// Mitsubishi GX Works2 project: PLC0918_V1   PLC: Q02/Q02H

PROGRAM MAIN
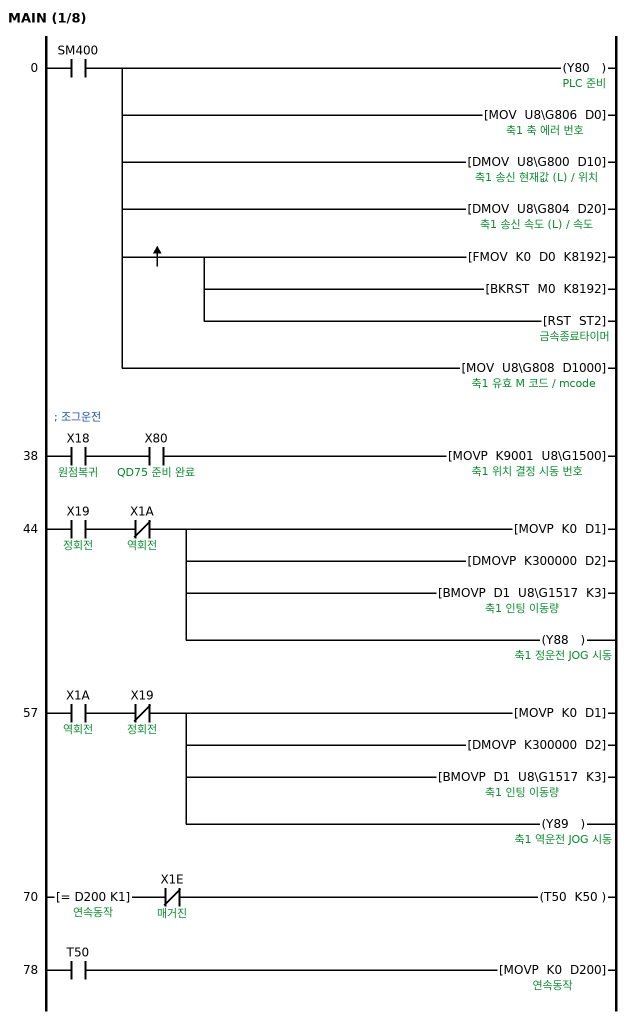
0     LD      SM400
      OUT     Y80  ; PLC 준비
      MOV     U8\G806 D0  ; 축1 축 에러 번호
      DMOV    U8\G800 D10  ; 축1 송신 현재값 (L) / 위치
      DMOV    U8\G804 D20  ; 축1 송신 속도 (L) / 속도
      MPS
      MEP
      FMOV    K0 D0 K8192
      BKRST   M0 K8192
      RST     ST2  ; 금속종료타이머
      MPP
      MOV     U8\G808 D1000  ; 축1 유효 M 코드 / mcode
; 조그운전
38    LD      X18  ; 원점복귀
      AND     X80  ; QD75 준비 완료
      MOVP    K9001 U8\G1500  ; 축1 위치 결정 시동 번호
44    LD      X19  ; 정회전
      ANI     X1A  ; 역회전
      MOVP    K0 D1
      DMOVP   K300000 D2
      BMOVP   D1 U8\G1517 K3  ; 축1 인팅 이동량
      OUT     Y88  ; 축1 정운전 JOG 시동
57    LD      X1A  ; 역회전
      ANI     X19  ; 정회전
      MOVP    K0 D1
      DMOVP   K300000 D2
      BMOVP   D1 U8\G1517 K3
      OUT     Y89  ; 축1 역운전 JOG 시동
70    LD=     D200 K1  ; 연속동작
      ANI     X1E  ; 매거진
      OUT     T50 K50
78    LD      T50
      MOVP    K0 D200
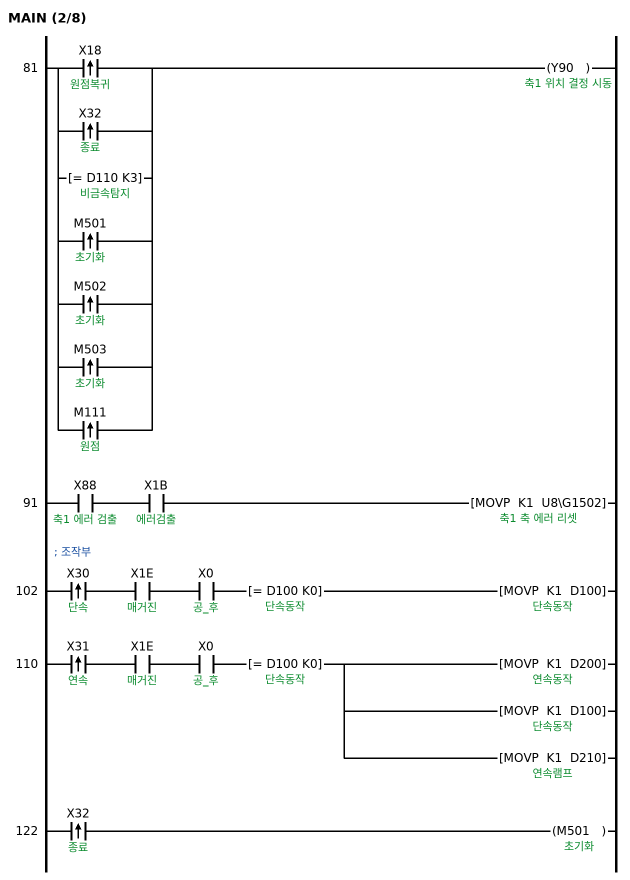
81    LDP     X18  ; 원점복귀
      ORP     X32  ; 종료
      OR=     D110 K3  ; 비금속탐지
      ORP     M501  ; 초기화
      ORP     M502  ; 초기화
      ORP     M503  ; 초기화
      ORP     M111  ; 원점
      OUT     Y90  ; 축1 위치 결정 시동
91    LD      X88  ; 축1 에러 검출
      AND     X1B  ; 에러검출
      MOVP    K1 U8\G1502  ; 축1 축 에러 리셋
; 조작부
102   LDP     X30  ; 단속
      AND     X1E  ; 매거진
      AND     X0  ; 공_후
      AND=    D100 K0  ; 단속동작
      MOVP    K1 D100
110   LDP     X31  ; 연속
      AND     X1E  ; 매거진
      AND     X0  ; 공_후
      AND=    D100 K0  ; 단속동작
      MOVP    K1 D200
      MOVP    K1 D100
      MOVP    K1 D210  ; 연속램프
122   LDP     X32  ; 종료
      OUT     M501  ; 초기화
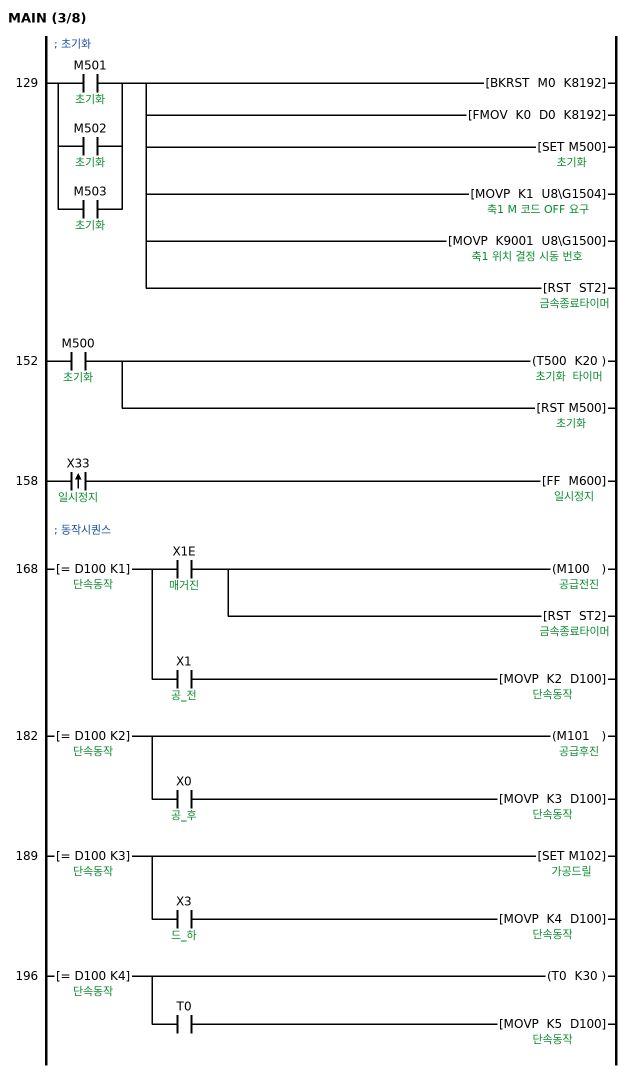
; 초기화
129   LD      M501  ; 초기화
      OR      M502  ; 초기화
      OR      M503  ; 초기화
      BKRST   M0 K8192
      FMOV    K0 D0 K8192
      SET     M500  ; 초기화
      MOVP    K1 U8\G1504  ; 축1 M 코드 OFF 요구
      MOVP    K9001 U8\G1500
      RST     ST2  ; 금속종료타이머
152   LD      M500  ; 초기화
      OUT     T500 K20  ; 초기화  타이머
      RST     M500  ; 초기화
158   LDP     X33  ; 일시정지
      FF      M600  ; 일시정지
; 동작시퀀스
168   LD=     D100 K1  ; 단속동작
      MPS
      AND     X1E  ; 매거진
      OUT     M100  ; 공급전진
      RST     ST2  ; 금속종료타이머
      MPP
      AND     X1  ; 공_전
      MOVP    K2 D100
182   LD=     D100 K2  ; 단속동작
      OUT     M101  ; 공급후진
      AND     X0  ; 공_후
      MOVP    K3 D100
189   LD=     D100 K3  ; 단속동작
      SET     M102  ; 가공드릴
      AND     X3  ; 드_하
      MOVP    K4 D100
196   LD=     D100 K4  ; 단속동작
      OUT     T0 K30
      AND     T0
      MOVP    K5 D100
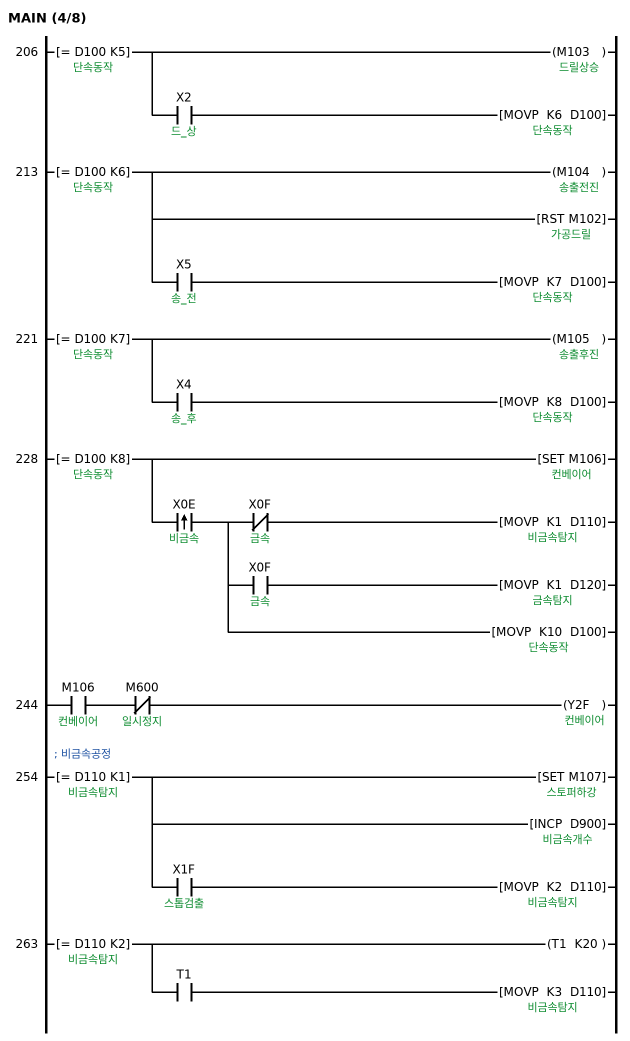
206   LD=     D100 K5  ; 단속동작
      OUT     M103  ; 드릴상승
      AND     X2  ; 드_상
      MOVP    K6 D100
213   LD=     D100 K6  ; 단속동작
      OUT     M104  ; 송출전진
      RST     M102  ; 가공드릴
      AND     X5  ; 송_전
      MOVP    K7 D100
221   LD=     D100 K7  ; 단속동작
      OUT     M105  ; 송출후진
      AND     X4  ; 송_후
      MOVP    K8 D100
228   LD=     D100 K8  ; 단속동작
      SET     M106  ; 컨베이어
      ANDP    X0E  ; 비금속
      MPS
      ANI     X0F  ; 금속
      MOVP    K1 D110
      MRD
      AND     X0F  ; 금속
      MOVP    K1 D120  ; 금속탐지
      MPP
      MOVP    K10 D100
244   LD      M106  ; 컨베이어
      ANI     M600  ; 일시정지
      OUT     Y2F  ; 컨베이어
; 비금속공정
254   LD=     D110 K1  ; 비금속탐지
      SET     M107  ; 스토퍼하강
      INCP    D900  ; 비금속개수
      AND     X1F  ; 스톱검출
      MOVP    K2 D110
263   LD=     D110 K2  ; 비금속탐지
      OUT     T1 K20
      AND     T1
      MOVP    K3 D110
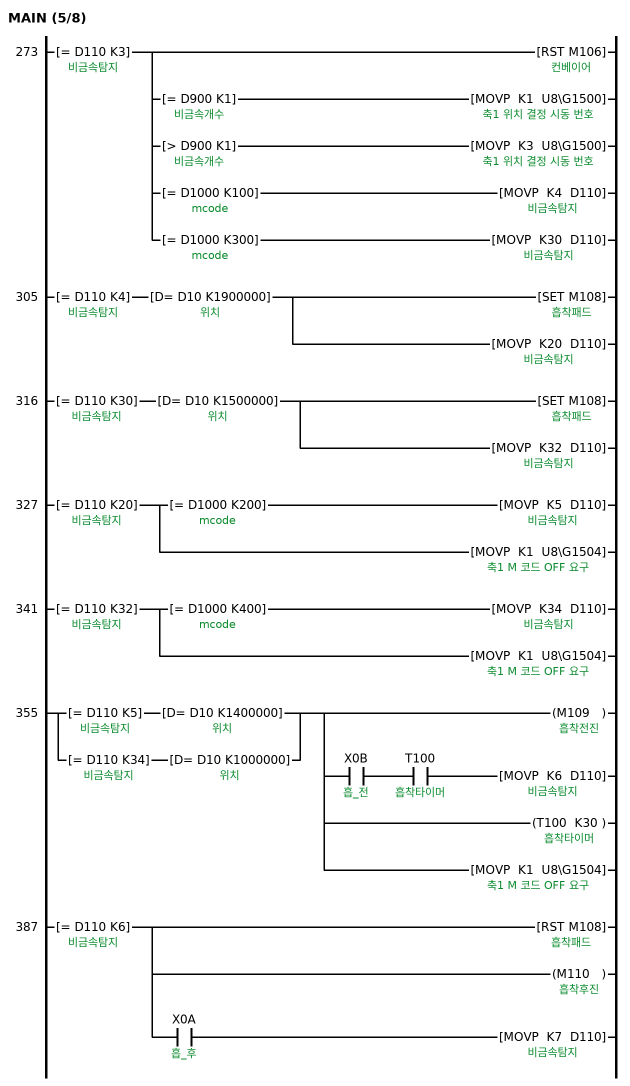
273   LD=     D110 K3  ; 비금속탐지
      RST     M106  ; 컨베이어
      MPS
      AND=    D900 K1  ; 비금속개수
      MOVP    K1 U8\G1500
      MRD
      AND>    D900 K1  ; 비금속개수
      MOVP    K3 U8\G1500
      MRD
      AND=    D1000 K100  ; mcode
      MOVP    K4 D110
      MPP
      AND=    D1000 K300  ; mcode
      MOVP    K30 D110
305   LD=     D110 K4  ; 비금속탐지
      ANDD=   D10 K1900000  ; 위치
      SET     M108  ; 흡착패드
      MOVP    K20 D110
316   LD=     D110 K30  ; 비금속탐지
      ANDD=   D10 K1500000  ; 위치
      SET     M108  ; 흡착패드
      MOVP    K32 D110
327   LD=     D110 K20  ; 비금속탐지
      MPS
      AND=    D1000 K200  ; mcode
      MOVP    K5 D110
      MPP
      MOVP    K1 U8\G1504
341   LD=     D110 K32  ; 비금속탐지
      MPS
      AND=    D1000 K400  ; mcode
      MOVP    K34 D110
      MPP
      MOVP    K1 U8\G1504
355   LD=     D110 K5  ; 비금속탐지
      ANDD=   D10 K1400000  ; 위치
      LD=     D110 K34  ; 비금속탐지
      ANDD=   D10 K1000000  ; 위치
      ORB
      OUT     M109  ; 흡착전진
      MPS
      AND     X0B  ; 흡_전
      AND     T100  ; 흡착타이머
      MOVP    K6 D110
      MPP
      OUT     T100 K30  ; 흡착타이머
      MOVP    K1 U8\G1504
387   LD=     D110 K6  ; 비금속탐지
      RST     M108  ; 흡착패드
      OUT     M110  ; 흡착후진
      AND     X0A  ; 흡_후
      MOVP    K7 D110
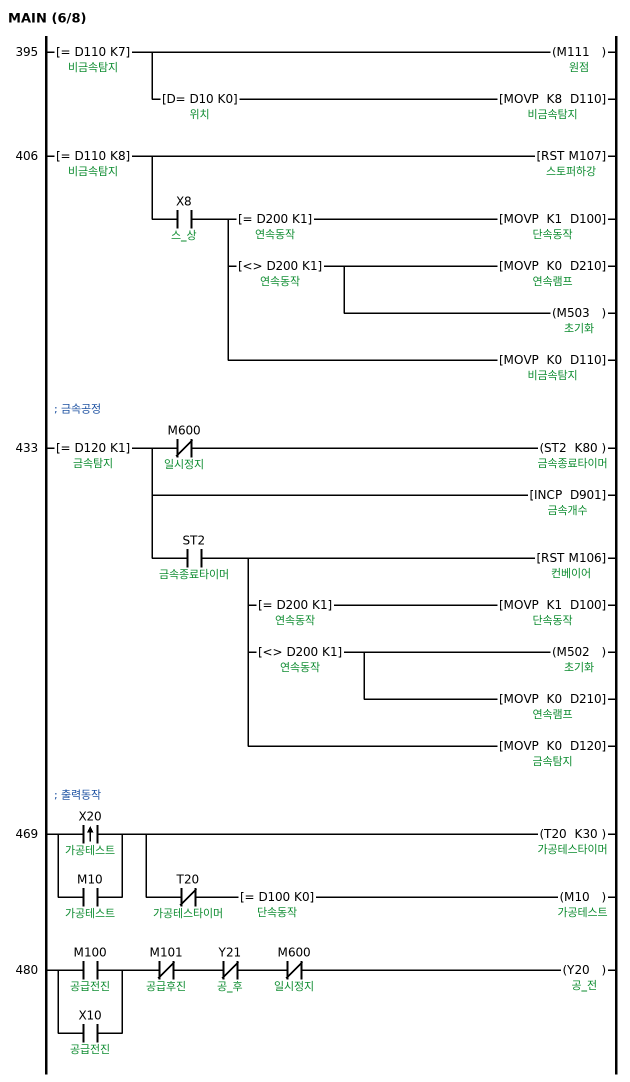
395   LD=     D110 K7  ; 비금속탐지
      OUT     M111  ; 원점
      ANDD=   D10 K0  ; 위치
      MOVP    K8 D110
406   LD=     D110 K8  ; 비금속탐지
      RST     M107  ; 스토퍼하강
      AND     X8  ; 스_상
      MPS
      AND=    D200 K1  ; 연속동작
      MOVP    K1 D100
      MRD
      AND<>   D200 K1  ; 연속동작
      MOVP    K0 D210
      OUT     M503  ; 초기화
      MPP
      MOVP    K0 D110
; 금속공정
433   LD=     D120 K1  ; 금속탐지
      MPS
      ANI     M600  ; 일시정지
      OUT     ST2 K80  ; 금속종료타이머
      MPP
      INCP    D901  ; 금속개수
      AND     ST2  ; 금속종료타이머
      RST     M106  ; 컨베이어
      MPS
      AND=    D200 K1  ; 연속동작
      MOVP    K1 D100
      MRD
      AND<>   D200 K1  ; 연속동작
      OUT     M502  ; 초기화
      MOVP    K0 D210
      MPP
      MOVP    K0 D120
; 출력동작
469   LDP     X20  ; 가공테스트
      OR      M10  ; 가공테스트
      OUT     T20 K30  ; 가공테스타이머
      ANI     T20  ; 가공테스타이머
      AND=    D100 K0  ; 단속동작
      OUT     M10  ; 가공테스트
480   LD      M100  ; 공급전진
      OR      X10  ; 공급전진
      ANI     M101  ; 공급후진
      ANI     Y21  ; 공_후
      ANI     M600  ; 일시정지
      OUT     Y20  ; 공_전
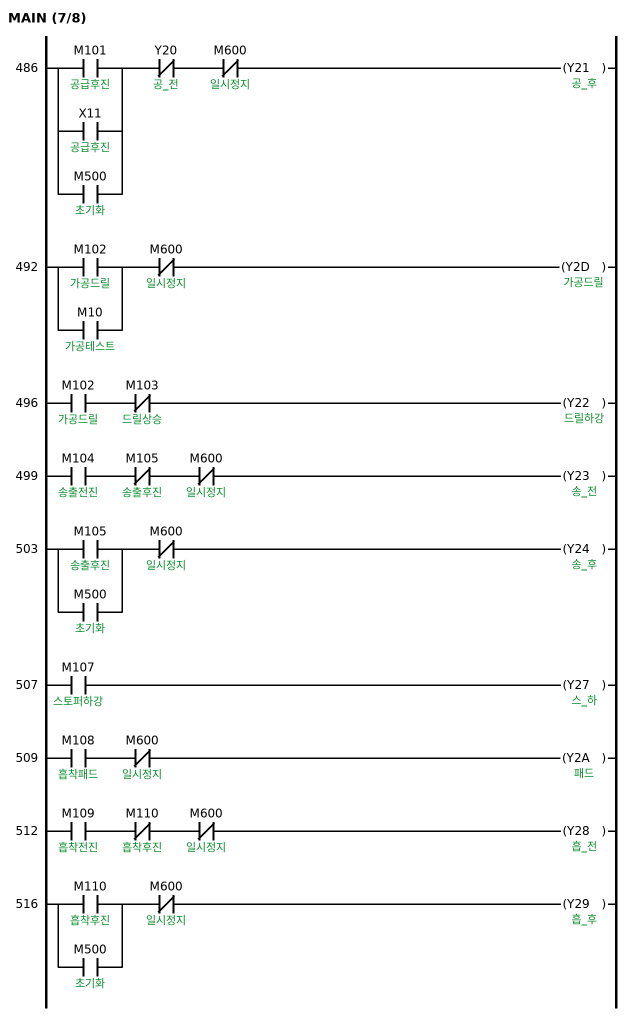
486   LD      M101  ; 공급후진
      OR      X11  ; 공급후진
      OR      M500  ; 초기화
      ANI     Y20  ; 공_전
      ANI     M600  ; 일시정지
      OUT     Y21  ; 공_후
492   LD      M102  ; 가공드릴
      OR      M10  ; 가공테스트
      ANI     M600  ; 일시정지
      OUT     Y2D  ; 가공드릴
496   LD      M102  ; 가공드릴
      ANI     M103  ; 드릴상승
      OUT     Y22  ; 드릴하강
499   LD      M104  ; 송출전진
      ANI     M105  ; 송출후진
      ANI     M600  ; 일시정지
      OUT     Y23  ; 송_전
503   LD      M105  ; 송출후진
      OR      M500  ; 초기화
      ANI     M600  ; 일시정지
      OUT     Y24  ; 송_후
507   LD      M107  ; 스토퍼하강
      OUT     Y27  ; 스_하
509   LD      M108  ; 흡착패드
      ANI     M600  ; 일시정지
      OUT     Y2A  ; 패드
512   LD      M109  ; 흡착전진
      ANI     M110  ; 흡착후진
      ANI     M600  ; 일시정지
      OUT     Y28  ; 흡_전
516   LD      M110  ; 흡착후진
      OR      M500  ; 초기화
      ANI     M600  ; 일시정지
      OUT     Y29  ; 흡_후
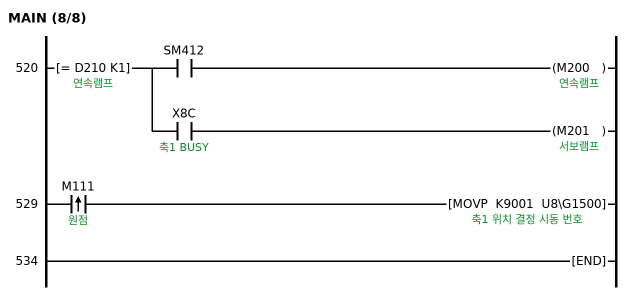
520   LD=     D210 K1  ; 연속램프
      MPS
      AND     SM412
      OUT     M200  ; 연속램프
      MPP
      AND     X8C  ; 축1 BUSY
      OUT     M201  ; 서보램프
529   LDP     M111  ; 원점
      MOVP    K9001 U8\G1500
534   END
END_PROGRAM

PROGRAM test2
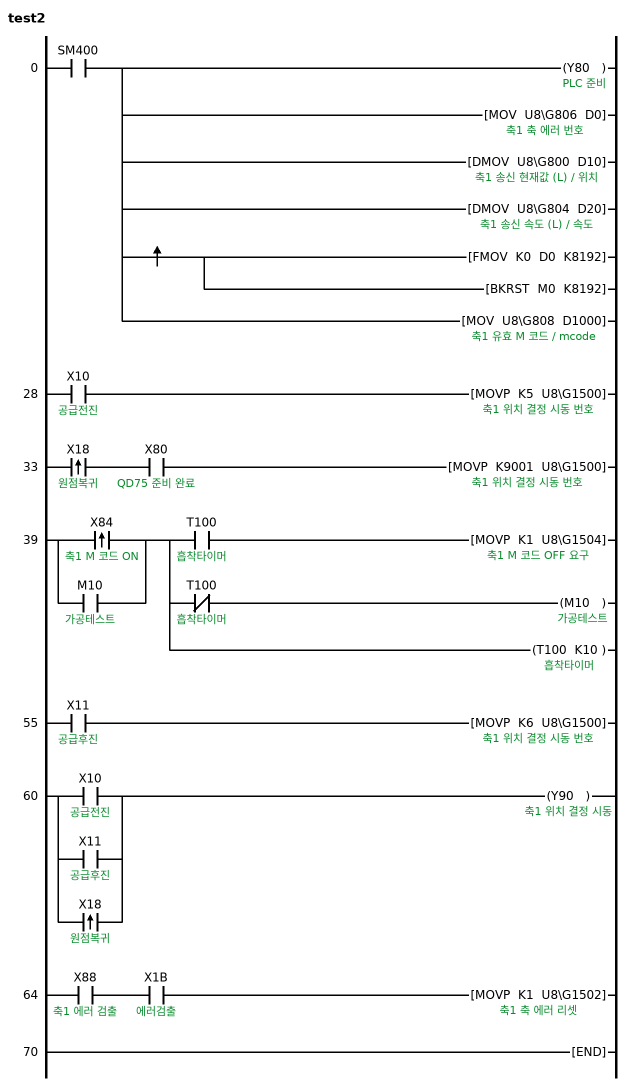
0     LD      SM400
      OUT     Y80  ; PLC 준비
      MOV     U8\G806 D0  ; 축1 축 에러 번호
      DMOV    U8\G800 D10  ; 축1 송신 현재값 (L) / 위치
      DMOV    U8\G804 D20  ; 축1 송신 속도 (L) / 속도
      MPS
      MEP
      FMOV    K0 D0 K8192
      BKRST   M0 K8192
      MPP
      MOV     U8\G808 D1000  ; 축1 유효 M 코드 / mcode
28    LD      X10  ; 공급전진
      MOVP    K5 U8\G1500  ; 축1 위치 결정 시동 번호
33    LDP     X18  ; 원점복귀
      AND     X80  ; QD75 준비 완료
      MOVP    K9001 U8\G1500
39    LDP     X84  ; 축1 M 코드 ON
      OR      M10  ; 가공테스트
      MPS
      AND     T100  ; 흡착타이머
      MOVP    K1 U8\G1504  ; 축1 M 코드 OFF 요구
      MRD
      ANI     T100  ; 흡착타이머
      OUT     M10  ; 가공테스트
      MPP
      OUT     T100 K10  ; 흡착타이머
55    LD      X11  ; 공급후진
      MOVP    K6 U8\G1500
60    LD      X10  ; 공급전진
      OR      X11  ; 공급후진
      ORP     X18  ; 원점복귀
      OUT     Y90  ; 축1 위치 결정 시동
64    LD      X88  ; 축1 에러 검출
      AND     X1B  ; 에러검출
      MOVP    K1 U8\G1502  ; 축1 축 에러 리셋
70    END
END_PROGRAM

PROGRAM OUTPUT
0     END
END_PROGRAM

// device comments not shown above
X6  ; 배_후
X7  ; 배_전
X9  ; 스_하
X0C  ; 창_후
X0D  ; 창_전
X21  ; 에러검출
X40  ; 원점복귀
X41  ; 정회전
X42  ; 역회전
X43  ; 에러검출
X81  ; 동기용 플래그
X85  ; 축2 M 코드 ON
X89  ; 축2 에러 검출
X8D  ; 축2 BUSY
X90  ; 축1 시동 완료
X91  ; 축2 시동 완료
X94  ; 축1 위치 결정 완료
X95  ; 축2 위치 결정 완료
Y25  ; 배_전
Y26  ; 배_후
Y2B  ; 창_전
Y2C  ; 창_후
Y84  ; 축1 축 정지
Y85  ; 축2 축 정지
Y8A  ; 축2 정운전 JOG 시동
Y8B  ; 축2 역운전 JOG 시동
Y91  ; 축2 위치 결정 시동
Y94  ; 축1 실행 금지 플래그
Y95  ; 축2 실행 금지 플래그
M150  ; 비금속타이머
T150  ; 비금속타이머
